(* IEC 61131-3 sources: eCockpitGit/test_project/src/%F%00 Library/%F%Common Functions/%F%String/%F%Big Input, 5 files *)

(* ---- %POU%FU_CheckNumberBI.st ---- *)
//This function checks if a string only contains numbers, dot (.) and dash (-) are also permitted as they are required for some numbers
//Returns true if string only contains numbers
// |**Version**|**Author**| **Date** |**Changes**
// | 1         | NSN      | 10-12-18 | Creation
FUNCTION FU_CheckNumberBI : BOOL
VAR_IN_OUT
	str			:STRING(1);	//String
END_VAR
VAR
	pStr		:POINTER TO BYTE;	//Address of source string
END_VAR
(*%!%__DELIMITER__%!%*)
pStr					:=		ADR(str);	//Address of source string
//It runs until string ends
WHILE pStr^ <> 0 DO
	//This checks if the selected character is in the range of numbers
	IF NOT((pStr^ >= 48 AND pStr^ <= 57) OR pStr^ = 46 OR pStr^ = 45) THEN
		RETURN;
	END_IF
	pStr				:=		pStr + 1;
END_WHILE
FU_CheckNumberBI		:=		TRUE;

(* ---- %POU%FU_OnlyNumbersBI.st ---- *)
//This function deletes all the none number characters from the string, until it finds zero
// |**Version**|**Author**| **Date** |**Changes**
// | 1         | NSN      | 19-06-18 | Creation
FUNCTION FU_OnlyNumbersBI
VAR_INPUT
	str			:STRING(1);			//String
END_VAR
VAR
	pStr		:POINTER TO BYTE := ADR(str);	//Address of source string
	StrBuff		:POINTER TO BYTE;	//Buffer for Address of the string
END_VAR
(*%!%__DELIMITER__%!%*)
IF pStr <> 0 THEN
	//Buffers are updated
	StrBuff					:=		pStr;
	//It runs until string ends
	WHILE pStr^ <> 0 DO
		//If a non number character is found, the next number character is then found
		WHILE StrBuff^ < EASCII.Zero OR StrBuff^ > EASCII.Nine DO
			//If no number is found before string end, it finishes
			IF StrBuff^ = 0 THEN
				pStr^		:=		0;
				RETURN;
			END_IF
			StrBuff			:=		StrBuff + 1;
		END_WHILE
		//Found number is copied
		pStr^				:=		StrBuff^;
		//Next character
		pStr				:=		pStr + 1;
		StrBuff				:=		StrBuff + 1;
	END_WHILE
END_IF

(* ---- %POU%FU_sCompareCaseInsensitive.st ---- *)
//This function compares two strings and ignores case
// Eg. Test = test is true
// |**Version**|**Author**| **Date** |**Changes**
// | 1         | NSN      | 08-03-22 | Creation
FUNCTION FU_sCompareCaseInsensitive : BOOL
VAR_IN_OUT
	s1			:STRING(1);			//Input String1
	s2			:STRING(1);			//Input String2
END_VAR
VAR
	i			:WORD;
	s1pb		:POINTER TO EASCII;
	s2pb		:POINTER TO EASCII;
END_VAR
(*%!%__DELIMITER__%!%*)
s1pb			:=		ADR(s1);
s2pb			:=		ADR(s2);
WHILE TRUE DO
	IF s1pb^ = 0 AND s2pb^ = 0 THEN
		FU_sCompareCaseInsensitive		:=		TRUE;
		RETURN;
	ELSIF s1pb^ <> s2pb^ THEN
		IF NOT(FU_bCompareCharCaseInsensitive(char1:=s1pb^,char2:=s2pb^)) THEN
			RETURN;
		END_IF
	END_IF
	s2pb		:=		s2pb + 1;
	s1pb		:=		s1pb + 1;
END_WHILE

(* ---- %POU%FU_sCopyBI.st ---- *)
//This functions copies the contents of one string into another (s1 to s2)
//It stops when string 1 ends
// |**Version**|**Author**| **Date** |**Changes**
// | 1         | NSN      | 05-02-19 | Creation
FUNCTION FU_sCopyBI
VAR_IN_OUT
	s1			:STRING(1);			//Input String1
	s2			:STRING(1);			//Input String2
END_VAR
VAR_INPUT
	s2MaxSize	:DWORD;
END_VAR
VAR
	s1pb		:POINTER TO BYTE;
	s2pb		:POINTER TO BYTE;
END_VAR
(*%!%__DELIMITER__%!%*)
s1pb			:=		ADR(s1);
s2pb			:=		ADR(s2);
WHILE TRUE DO
	IF s1pb^ = 0 OR s2MaxSize = 0 THEN
		RETURN;
	END_IF
	s2pb^		:=		s1pb^;
	s2pb		:=		s2pb + 1;
	s1pb		:=		s1pb + 1;
	s2MaxSize	:=		s2MaxSize - 1;
END_WHILE

(* ---- %POU%FU_sDecTruncBI.st ---- *)
//This function, limits the amount of decimals after the decimal point, the decimal point is the english .
// +-----------+----------+----------+-----------------------------------------------------------------------------------------------------------------------+
// |**Version**|**Author**| **Date** |**Changes**                                                                                                            |
// +-----------+----------+----------+-----------------------------------------------------------------------------------------------------------------------+
// | 1         | NSN      | 29-01-19 | Creation                                                                                                              |
// +-----------+----------+----------+-----------------------------------------------------------------------------------------------------------------------+
FUNCTION FU_sDecTruncBI : BOOL
VAR_IN_OUT
	str			:STRING(1);			//Input String
END_VAR
VAR_INPUT
	decimals	:WORD;				//How many decimals should be kept
END_VAR
VAR_INPUT
	pStr		:POINTER TO BYTE := ADR(str);	//Address of the string
END_VAR
(*%!%__DELIMITER__%!%*)
IF pStr <> 0 THEN
	WHILE pStr^ <> EASCII.Dot DO
		IF pStr^ = 0 THEN
			RETURN;
		END_IF
		pStr			:=		pStr + 1;
	END_WHILE
	IF decimals = 0 THEN
		pStr^			:=		0;
		RETURN;
	ELSE
		decimals		:=		decimals + 1;
		WHILE pStr^ <> 0 AND decimals > 0 DO
			pStr		:=		pStr + 1;
			decimals	:=		decimals - 1;
		END_WHILE
		pStr^			:=		0;
		RETURN;
	END_IF
END_IF
